(*
    FB_SaveCalibrationReport
    - One-shot wrapper: builds the calibration JSON and writes it to disk.
*)
FUNCTION_BLOCK FB_SaveCalibrationReport
VAR_INPUT
	bExecute            : BOOL;  // Rising edge starts the build+save sequence
    sUser               : STRING(64);

    stReportInfo        : ST_ReportInfo;
    stCalibrationInfo   : ST_CalibrationInfo;
    aCalibrationData    : ARRAY[1..250] OF ST_CalibrationData;
    iDataCount          : INT;   // Valid range: 0..100 (0 allowed -> empty list)
END_VAR
VAR_OUTPUT
	bDone       : BOOL;          // TRUE when file is saved and closed
    bBusy       : BOOL;          // TRUE while internal state machine is running
    bError      : BOOL;          // TRUE on any error
    nErrId      : UDINT;         // Error code propagated from child FBs
    sFileNameOut: STRING(256);   // Full path of the output JSON file
END_VAR
VAR
	// State machine
    iStep       : INT;           // 0=IDLE, 10=BUILD, 20=SAVE, 100=LATCH

    // Edge detection for bExecute
    rtExec      : R_TRIG;

    // Child FBs
    fbBuild     : FB_BuildCalReportJson;
    fbSave      : FB_SaveCalReportToFile;

    // Buffer for JSON document produced by builder
    sBuf        : STRING(16384);
	nBufBytes 	: UDINT;          // <- NEW
END_VAR

// --------------------------- IMPLEMENTATION ----------------------------------
rtExec(CLK := bExecute);

CASE iStep OF
    // -------------------------------------------------------------------------
    0: // IDLE: arm on rising edge of bExecute
    // -------------------------------------------------------------------------
    IF rtExec.Q THEN
        // Clamp iDataCount to valid limits (defensive)
        IF iDataCount < 0   THEN iDataCount := 0;   END_IF;
        IF iDataCount > 100 THEN iDataCount := 100; END_IF;

        // Clear latched outputs and mark busy
        bDone := FALSE; bError := FALSE; nErrId := 0;
        sFileNameOut := '';
        bBusy := TRUE;

        // Jump to build step
        iStep := 10;
    END_IF

    // -------------------------------------------------------------------------
    10: // BUILD JSON: FB_BuildCalReportJson (single-shot)
    // -------------------------------------------------------------------------
    fbBuild(
        stReportInfo      := stReportInfo,
        stCalibrationInfo := stCalibrationInfo,
        aCalibrationData  := aCalibrationData,
		iCalNumber  	  := TO_INT(stCalibrationInfo.iCalibrationNumber),
		sUser        	  := sUser,
        iDataCount        := iDataCount
    );

    IF fbBuild.bDone THEN
        // Copy the produced JSON document into our local buffer
        sBuf      := fbBuild.sJsonBuffer;
		nBufBytes := fbBuild.nJsonBytes;
		sFileNameOut := fbBuild.sFileNameOut;

        // Proceed to SAVE step
        iStep := 20;

    ELSIF fbBuild.bError THEN
        // Propagate error and latch
        bError := TRUE;
        nErrId := fbBuild.nErrId;
        bBusy := FALSE;
        iStep := 100;
    END_IF

    // -------------------------------------------------------------------------
    20: // SAVE FILE: FB_SaveCalReportToFile (stateful)
    // -------------------------------------------------------------------------
    
	fbSave(
        bExecute    := TRUE,  // keep TRUE while we wait for bDone/bError
        sJsonBuffer := sBuf,
		nJsonBytes  := nBufBytes,
		sFileNameIn := sFileNameOut,
    );

    IF fbSave.bDone THEN
        bDone := TRUE;
        bBusy := FALSE;
        iStep := 100;

    ELSIF fbSave.bError THEN
        bError := TRUE;
        nErrId := fbSave.nErrId;
        bBusy := FALSE;
        iStep := 100;
    END_IF

    // -------------------------------------------------------------------------
    100: // LATCH: wait caller to drop bExecute to return to IDLE
    // -------------------------------------------------------------------------
    // Keep driving fbSave with bExecute := FALSE to let it reset internally.
    fbSave(bExecute := FALSE);

    IF NOT bExecute THEN
        // Return to IDLE after caller drops the trigger
        iStep := 0;
    END_IF
END_CASE

METHOD Reset : BOOL
VAR_INPUT
END_VAR
// Latch outputs & codes
bDone        := FALSE;
bBusy        := FALSE;
bError       := FALSE;
nErrId       := 0;
sFileNameOut := '';

// State machine
iStep := 0;

// Internal buffers
sBuf      := '';
nBufBytes := 0;

// Politely reset child FBs (if their Reset() exists; otherwise just de-assert)
fbBuild.Reset(); // returns TRUE/ignored; leaves builder idle
fbSave.Reset();  // returns TRUE/ignored; leaves saver idle

// Extra safety: ensure no lingering executes this cycle
fbSave(bExecute := FALSE);

Reset := TRUE;
END_METHOD

END_FUNCTION_BLOCK

(* stored: Version 1.1.0.1, ProductVersion 3.1.4024.15
   POU FB_SaveCalibrationReport: Id {a5055892-3336-4cd7-b90e-e7e659f72c7e}, SpecialFunc None
   Method Reset: Id {c32e696b-e79a-4aaf-b674-1619dcf03194} *)
